FUNCTION_BLOCK String_Test EXTENDS TcUnit.FB_TestSuite
VAR_INPUT
END_VAR
VAR_OUTPUT
END_VAR
VAR
END_VAR

END_FUNCTION_BLOCK

(* stored: Version 1.1.0.1
   POU String_Test: Id {9a42e009-eb20-4d8c-bcd8-047061b12bfc}, SpecialFunc None *)
